PROGRAM HRL_SkillSet
VAR
//Hochregallager Skillset	
	
	//HRL Conveyorbelt Skills
	{attribute 'OPC.UA.DA':= '1'}
	HRL_Skill_CB_MoveForwards: HRL_CB_AS_HorizontalMove; //Movement to Store-Out some goods on the Conveyorbelt
	{attribute 'OPC.UA.DA':= '1'}
	HRL_Skill_CB_MoveBackwards : HRL_CB_AS_HorizontalMove; //Movement to Store-In some goods on the Conveyorbelt
	
	//HRL RGB Skills
	{attribute 'OPC.UA.DA':= '1'}
	HRL_Skill_RGB_MoveBackwards : HRL_RGB_AS_HorizontalMoveSensors;	
	{attribute 'OPC.UA.DA':= '1'}
	HRL_Skill_RGB_MoveForwards : HRL_RGB_AS_HorizontalMoveSensors;	
	{attribute 'OPC.UA.DA':= '1'}
	HRL_Skill_RGB_MoveVerticalForwards : HRL_RGB_AS_VerticalMoveEncoder;	
	{attribute 'OPC.UA.DA':= '1'}
	HRL_Skill_RGB_MoveVerticalBackwards : HRL_RGB_AS_VerticalMoveEncoder;
	{attribute 'OPC.UA.DA':= '1'}
	HRL_Skill_RGB_MoveHorizontalForwards : HRL_RGB_AS_HorizontalMoveEncoder;	
	{attribute 'OPC.UA.DA':= '1'}
	HRL_Skill_RGB_MoveHorizontalBackwards : HRL_RGB_AS_HorizontalMoveEncoder;
	
	HRL_ControlOfOutputs : HRL_COntrolOfOutputs;
	HRL_OperatingModes : HRL_OperatingModes;
//TestMethode NMethode für Auslagern //
	{attribute 'OPC.UA.DA':= '1'}
	HRL_NMethod_Auslagern :HRL_NMethod_Auslagern;

//Variablensetzung: Sollte später über SkillOA eingesetzt werden ODER Hard in SPS codiert (Diskussionspunkt)
	TIME_TSR : TIME := T#150MS;
	ResetButton: BOOL;
	StartButton: BOOL;
	ConfirmationButton: BOOL;
END_VAR

VAR_OUTPUT
	HRL_CB_forwards : BOOL; //GVL_HRL.HRL_MOT_Foerderband_vorwaerts
	HRL_CB_backwards : BOOL; //GVL_HRL.HRL_MOT_Foerderband_rueckwaerts
	HRL_RGB_Forwards01 : BOOL; //GVL_HRL.HRL_MOT_Ausleger_vorwaerts
	HRL_RGB_Forwards02 : BOOL; //GVL_HRL.HRL_MOT_Ausleger_rueckwaerts
	HRL_RGB_Backwards01 : BOOL; //GVL_HRL.HRL_MOT_Ausleger_rueckwaerts
	HRL_RGB_Backwards02 : BOOL; //GVL_HRL.HRL_MOT_Ausleger_vorwaerts
	HRL_RGB_VertikalDown01 : BOOL; //GVL_HRL.HRL_MOT_vertikal_runter
	HRL_RGB_VertikalDown02 : BOOL; //GVL_HRL.HRL_MOT_vertikal_hoch
	HRL_RGB_VertikalUp01 : BOOL; //GVL_HRL.HRL_MOT_vertikal_hoch
	HRL_RGB_VertikalUp02 : BOOL; //GVL_HRL.HRL_MOT_vertikal_runter
	HRL_RGB_HorizontalForwards01 : BOOL; //GVL_HRL.HRL_MOT_horizontal_zum_Regal
	HRL_RGB_HorizontalForwards02 : BOOL; //GVL_HRL.HRL_MOT_horizontal_zum_Foerderband
	HRL_RGB_HorizontalBackwards01 : BOOL; //GVL_HRL.HRL_MOT_horizontal_zum_Foerderband
	HRL_RGB_HorizontalBackwards02 : BOOL; //GVL_HRL.HRL_MOT_horizontal_zum_Regal
END_VAR

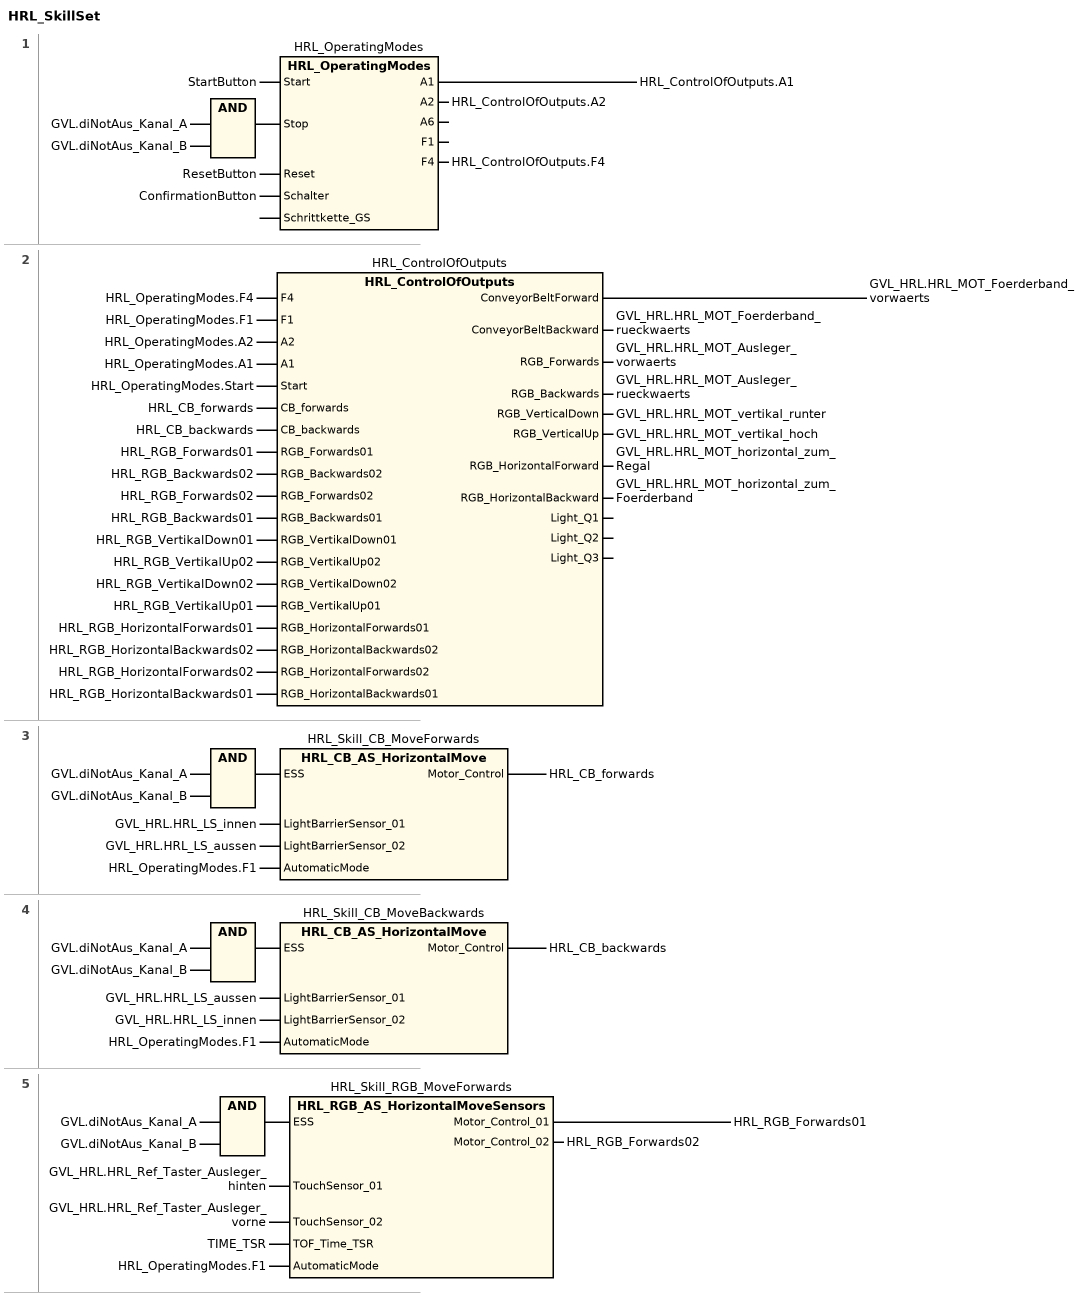
// NETWORK 1
HRL_OperatingModes(
    Start := StartButton,
    Stop := GVL.diNotAus_Kanal_A AND GVL.diNotAus_Kanal_B,
    Reset := ResetButton,
    Schalter := ConfirmationButton,
    A2 => HRL_ControlOfOutputs.A2,
    F4 => HRL_ControlOfOutputs.F4);
HRL_ControlOfOutputs.A1 := HRL_OperatingModes.A1;

// NETWORK 2
HRL_ControlOfOutputs(
    F4 := HRL_OperatingModes.F4,
    F1 := HRL_OperatingModes.F1,
    A2 := HRL_OperatingModes.A2,
    A1 := HRL_OperatingModes.A1,
    Start := HRL_OperatingModes.Start,
    CB_forwards := HRL_CB_forwards,
    CB_backwards := HRL_CB_backwards,
    RGB_Forwards01 := HRL_RGB_Forwards01,
    RGB_Backwards02 := HRL_RGB_Backwards02,
    RGB_Forwards02 := HRL_RGB_Forwards02,
    RGB_Backwards01 := HRL_RGB_Backwards01,
    RGB_VertikalDown01 := HRL_RGB_VertikalDown01,
    RGB_VertikalUp02 := HRL_RGB_VertikalUp02,
    RGB_VertikalDown02 := HRL_RGB_VertikalDown02,
    RGB_VertikalUp01 := HRL_RGB_VertikalUp01,
    RGB_HorizontalForwards01 := HRL_RGB_HorizontalForwards01,
    RGB_HorizontalBackwards02 := HRL_RGB_HorizontalBackwards02,
    RGB_HorizontalForwards02 := HRL_RGB_HorizontalForwards02,
    RGB_HorizontalBackwards01 := HRL_RGB_HorizontalBackwards01,
    ConveyorBeltBackward => GVL_HRL.HRL_MOT_Foerderband_rueckwaerts,
    RGB_Forwards => GVL_HRL.HRL_MOT_Ausleger_vorwaerts,
    RGB_Backwards => GVL_HRL.HRL_MOT_Ausleger_rueckwaerts,
    RGB_VerticalDown => GVL_HRL.HRL_MOT_vertikal_runter,
    RGB_VerticalUp => GVL_HRL.HRL_MOT_vertikal_hoch,
    RGB_HorizontalForward => GVL_HRL.HRL_MOT_horizontal_zum_Regal,
    RGB_HorizontalBackward => GVL_HRL.HRL_MOT_horizontal_zum_Foerderband);
GVL_HRL.HRL_MOT_Foerderband_vorwaerts := HRL_ControlOfOutputs.ConveyorBeltForward;

// NETWORK 3
HRL_Skill_CB_MoveForwards(
    ESS := GVL.diNotAus_Kanal_A AND GVL.diNotAus_Kanal_B,
    LightBarrierSensor_01 := GVL_HRL.HRL_LS_innen,
    LightBarrierSensor_02 := GVL_HRL.HRL_LS_aussen,
    AutomaticMode := HRL_OperatingModes.F1); // HRL_CB_AS_HorizontalMove
HRL_CB_forwards := HRL_Skill_CB_MoveForwards.Motor_Control;

// NETWORK 4
HRL_Skill_CB_MoveBackwards(
    ESS := GVL.diNotAus_Kanal_A AND GVL.diNotAus_Kanal_B,
    LightBarrierSensor_01 := GVL_HRL.HRL_LS_aussen,
    LightBarrierSensor_02 := GVL_HRL.HRL_LS_innen,
    AutomaticMode := HRL_OperatingModes.F1); // HRL_CB_AS_HorizontalMove
HRL_CB_backwards := HRL_Skill_CB_MoveBackwards.Motor_Control;

// NETWORK 5
HRL_Skill_RGB_MoveForwards(
    ESS := GVL.diNotAus_Kanal_A AND GVL.diNotAus_Kanal_B,
    TouchSensor_01 := GVL_HRL.HRL_Ref_Taster_Ausleger_hinten,
    TouchSensor_02 := GVL_HRL.HRL_Ref_Taster_Ausleger_vorne,
    TOF_Time_TSR := TIME_TSR,
    AutomaticMode := HRL_OperatingModes.F1,
    Motor_Control_02 => HRL_RGB_Forwards02); // HRL_RGB_AS_HorizontalMoveSensors
HRL_RGB_Forwards01 := HRL_Skill_RGB_MoveForwards.Motor_Control_01;

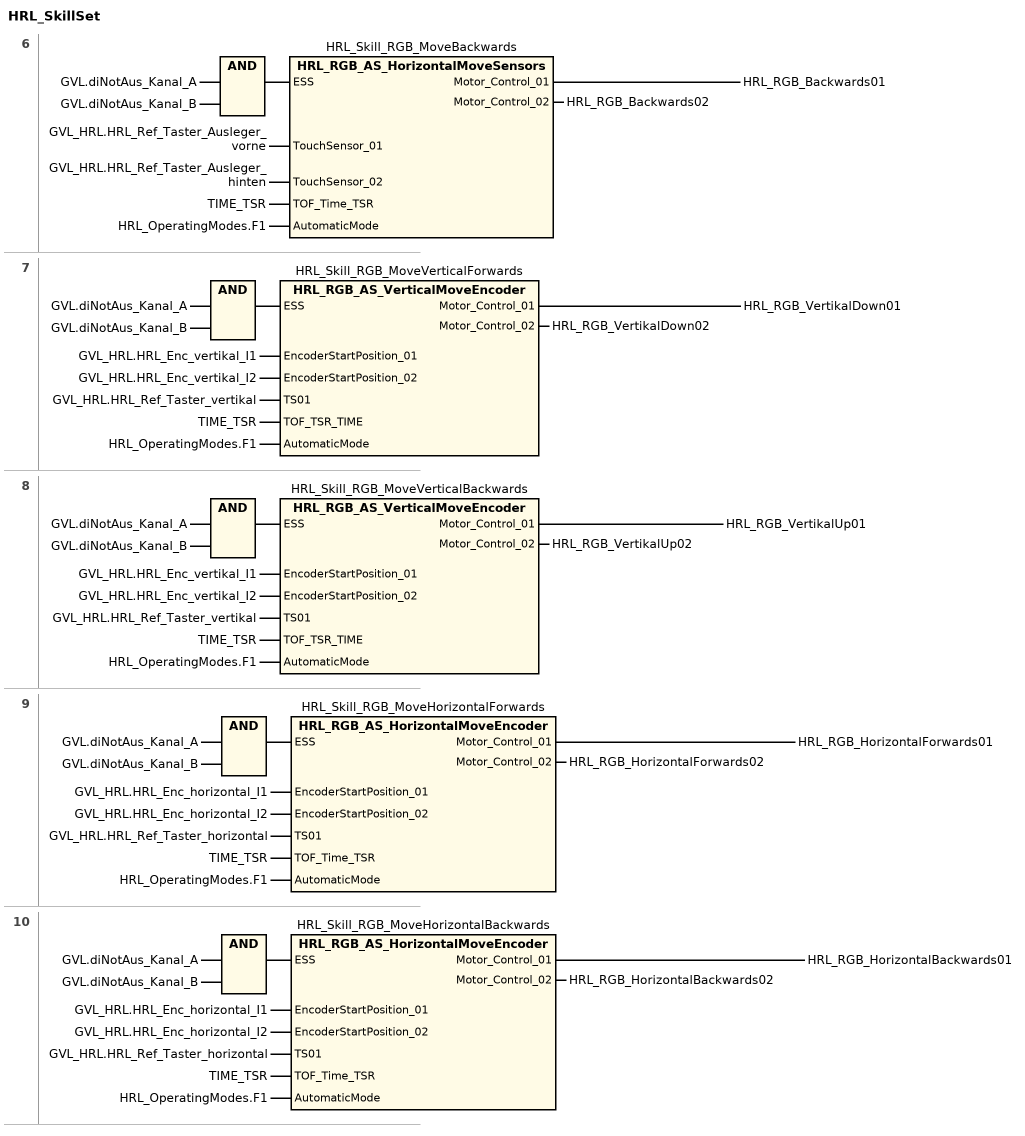
// NETWORK 6
HRL_Skill_RGB_MoveBackwards(
    ESS := GVL.diNotAus_Kanal_A AND GVL.diNotAus_Kanal_B,
    TouchSensor_01 := GVL_HRL.HRL_Ref_Taster_Ausleger_vorne,
    TouchSensor_02 := GVL_HRL.HRL_Ref_Taster_Ausleger_hinten,
    TOF_Time_TSR := TIME_TSR,
    AutomaticMode := HRL_OperatingModes.F1,
    Motor_Control_02 => HRL_RGB_Backwards02); // HRL_RGB_AS_HorizontalMoveSensors
HRL_RGB_Backwards01 := HRL_Skill_RGB_MoveBackwards.Motor_Control_01;

// NETWORK 7
HRL_Skill_RGB_MoveVerticalForwards(
    ESS := GVL.diNotAus_Kanal_A AND GVL.diNotAus_Kanal_B,
    EncoderStartPosition_01 := GVL_HRL.HRL_Enc_vertikal_I1,
    EncoderStartPosition_02 := GVL_HRL.HRL_Enc_vertikal_I2,
    TS01 := GVL_HRL.HRL_Ref_Taster_vertikal,
    TOF_TSR_TIME := TIME_TSR,
    AutomaticMode := HRL_OperatingModes.F1,
    Motor_Control_02 => HRL_RGB_VertikalDown02); // HRL_RGB_AS_VerticalMoveEncoder
HRL_RGB_VertikalDown01 := HRL_Skill_RGB_MoveVerticalForwards.Motor_Control_01;

// NETWORK 8
HRL_Skill_RGB_MoveVerticalBackwards(
    ESS := GVL.diNotAus_Kanal_A AND GVL.diNotAus_Kanal_B,
    EncoderStartPosition_01 := GVL_HRL.HRL_Enc_vertikal_I1,
    EncoderStartPosition_02 := GVL_HRL.HRL_Enc_vertikal_I2,
    TS01 := GVL_HRL.HRL_Ref_Taster_vertikal,
    TOF_TSR_TIME := TIME_TSR,
    AutomaticMode := HRL_OperatingModes.F1,
    Motor_Control_02 => HRL_RGB_VertikalUp02); // HRL_RGB_AS_VerticalMoveEncoder
HRL_RGB_VertikalUp01 := HRL_Skill_RGB_MoveVerticalBackwards.Motor_Control_01;

// NETWORK 9
HRL_Skill_RGB_MoveHorizontalForwards(
    ESS := GVL.diNotAus_Kanal_A AND GVL.diNotAus_Kanal_B,
    EncoderStartPosition_01 := GVL_HRL.HRL_Enc_horizontal_I1,
    EncoderStartPosition_02 := GVL_HRL.HRL_Enc_horizontal_I2,
    TS01 := GVL_HRL.HRL_Ref_Taster_horizontal,
    TOF_Time_TSR := TIME_TSR,
    AutomaticMode := HRL_OperatingModes.F1,
    Motor_Control_02 => HRL_RGB_HorizontalForwards02); // HRL_RGB_AS_HorizontalMoveEncoder
HRL_RGB_HorizontalForwards01 := HRL_Skill_RGB_MoveHorizontalForwards.Motor_Control_01;

// NETWORK 10
HRL_Skill_RGB_MoveHorizontalBackwards(
    ESS := GVL.diNotAus_Kanal_A AND GVL.diNotAus_Kanal_B,
    EncoderStartPosition_01 := GVL_HRL.HRL_Enc_horizontal_I1,
    EncoderStartPosition_02 := GVL_HRL.HRL_Enc_horizontal_I2,
    TS01 := GVL_HRL.HRL_Ref_Taster_horizontal,
    TOF_Time_TSR := TIME_TSR,
    AutomaticMode := HRL_OperatingModes.F1,
    Motor_Control_02 => HRL_RGB_HorizontalBackwards02); // HRL_RGB_AS_HorizontalMoveEncoder
HRL_RGB_HorizontalBackwards01 := HRL_Skill_RGB_MoveHorizontalBackwards.Motor_Control_01;

END_PROGRAM

(* stored: Version 1.1.0.1, ProductVersion 3.1.4024.15
   POU HRL_SkillSet: Id {2fc9da90-1326-4a7b-a7d0-39451b3dbdc6}, SpecialFunc None *)
